// Mitsubishi GX Works2 project: 0729금비금미완   PLC: Q02/Q02H

PROGRAM MAIN
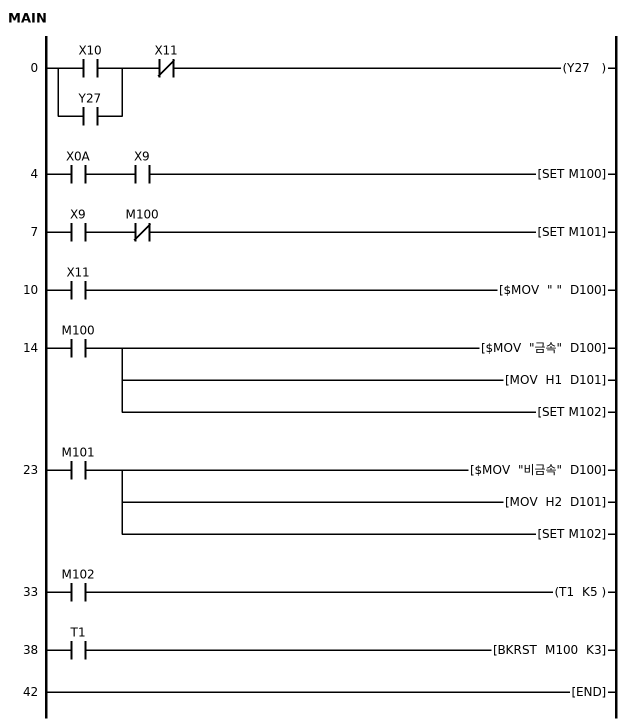
0     LD      X10
      OR      Y27
      ANI     X11
      OUT     Y27
4     LD      X0A
      AND     X9
      SET     M100
7     LD      X9
      ANI     M100
      SET     M101
10    LD      X11
      $MOV    "" D100
14    LD      M100
      $MOV    "금속" D100
      MOV     H1 D101
      SET     M102
23    LD      M101
      $MOV    "비금속" D100
      MOV     H2 D101
      SET     M102
33    LD      M102
      OUT     T1 K5
38    LD      T1
      BKRST   M100 K3
42    END
END_PROGRAM
